// TwinCAT 3 PLC project PLC01
// ProgramVersion: 3.1.4026.16
// CompilerDefines: VISU_USEPROPERTYINFO
// libraries:
//   Tc2_Standard, * (Beckhoff Automation GmbH)
//   Tc2_System, * (Beckhoff Automation GmbH)
//   Tc2_Utilities, * (Beckhoff Automation GmbH)
//   Tc3_EventLogger, * (Beckhoff Automation GmbH)
//   VisuElemEventTable, * (System)
// project tree:
//   / GlobalTextList.TcGTLO, PlcTask.TcTTO, Visualization Manager.TcVMO (not stored)
//   POUs/ MAIN.TcPOU, prgAlarmHnd.TcPOU
//   VISUs/ Footer.TcVIS, Visualization.TcVIS
// real-time tasks:
//   TASK PlcTask: cycle T#10ms, priority 20, ADS port 350

CONFIGURATION PLC01
    RESOURCE PLC ON TwinCAT3
        TASK PlcTask(INTERVAL := T#10ms, PRIORITY := 20);
        PROGRAM MAIN WITH PlcTask : MAIN;
    END_RESOURCE
END_CONFIGURATION

// ---- POUs/MAIN.TcPOU
PROGRAM MAIN
VAR
END_VAR


prgAlarmHnd();

END_PROGRAM

// ---- POUs/prgAlarmHnd.TcPOU
PROGRAM prgAlarmHnd
VAR
	evtReader: FB_ReadTc3Events;
	actualEvts: ARRAY[1..80] OF ST_ReadEventW;
	histEvts: ARRAY[1..80] OF ST_ReadEventW;
	doClearEvts, doConfirmEvts, doRaiseEvt1, doRaiseEvt2, doRaiseEvt3, doClearTable:BOOL;
	alarm1, alarm2, alarm3: FB_TcAlarm;
	hr, hrLastErr: HRESULT;
	raiseEvt1Trig, raiseEvt2Trig, raiseEvt3Trig:R_TRIG;
	clearEvt1Trig, clearEvt2Trig, clearEvt3Trig: F_TRIG;
	doInitNow:BOOL:=TRUE;
END_VAR

IF doInitNow THEN
	hr := alarm1.CreateEx(TC_Events.UserAlarms.evt01,TRUE,0);
	IF failed(hr) THEN
		hrLastErr:=hr;
	END_IF
	hr := alarm2.CreateEx(TC_Events.UserAlarms.evt02,TRUE,0);
	IF failed(hr) THEN
		hrLastErr:=hr;
	END_IF
	hr := alarm3.CreateEx(TC_Events.UserAlarms.evt03,TRUE,0);
	IF failed(hr) THEN
		hrLastErr:=hr;
	END_IF
	doInitNow:=FALSE;
END_IF
raiseEvt1Trig(CLK:= doRaiseEvt1);
raiseEvt2Trig(CLK:= doRaiseEvt2);
raiseEvt3Trig(CLK:= doRaiseEvt3 );
clearEvt1Trig(CLK:= doRaiseEvt1);
clearEvt2Trig(CLK:= doRaiseEvt2);
clearEvt3Trig(CLK:= doRaiseEvt3);

IF raiseEvt1Trig.Q THEN
	alarm1.Raise(0);
END_IF
IF raiseEvt2Trig.Q THEN
	alarm2.Raise(0);
END_IF
IF raiseEvt3trig.Q THEN
	alarm3.Raise(0);
END_IF
IF clearEvt1Trig.Q THEN
	alarm1.Clear(0,FALSE);
END_IF
IF clearEvt2Trig.Q THEN
	alarm2.Clear(0,FALSE);
END_IF
IF clearEvt3Trig.Q THEN
	alarm3.Clear(0,FALSE);
END_IF
IF doConfirmEvts THEN
	alarm1.Confirm(0);
	alarm2.Confirm(0);
	alarm3.Confirm(0);
END_IF

evtReader(
	bReadEvents:= TRUE, 
	nLanguageID:=1031 , 
	eDateAndTimeFormat:=E_DateAndTimeFormat.de_DE , 
	bClearTable:= doClearTable, 
	eMinSeverity:= , 
	aEvents=>actualEvts , 
	nNumberOfEvents=> , 
	bError=> , 
	hrErrorCode=> );

END_PROGRAM

// ---- GlobalTextList.TcGTLO
TEXTLIST GlobalTextList
  989 = 'Alarme 1'
  381 = 'Alarme 2'
  386 = 'Alarmes'
  56 = 'Classe'
  849 = 'Clear'
  728 = 'Confirma'
  493 = 'Confirmado'
  120 = 'Dara'
  682 = 'Data'
  44 = 'Fonte'
  901 = 'Histórico'
  39 = 'Hora'
  829 = 'Id'
  14 = 'Limpa'
  587 = 'Mensagem'
  374 = 'Origem'
  83 = 'srcId'
END_TEXTLIST

// ---- VISUs/Footer.TcVIS
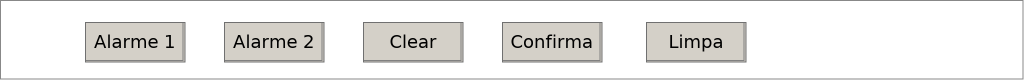
VISUALIZATION Footer  // 1024x80
    Button (85,22 100x40), "Alarme 1"
        toggle prgAlarmHnd.doRaiseEvt1
    Button (224,22 100x40), "Alarme 2"
        toggle prgAlarmHnd.doRaiseEvt2
    Button (363,22 100x40), "Clear"
        tap prgAlarmHnd.doClearEvts
    Button (502,22 100x40), "Confirma"
        tap prgAlarmHnd.doConfirmEvts
    Button (646,22 100x40), "Limpa"
        tap prgAlarmHnd.doClearTable
END_VISUALIZATION

// ---- VISUs/Visualization.TcVIS
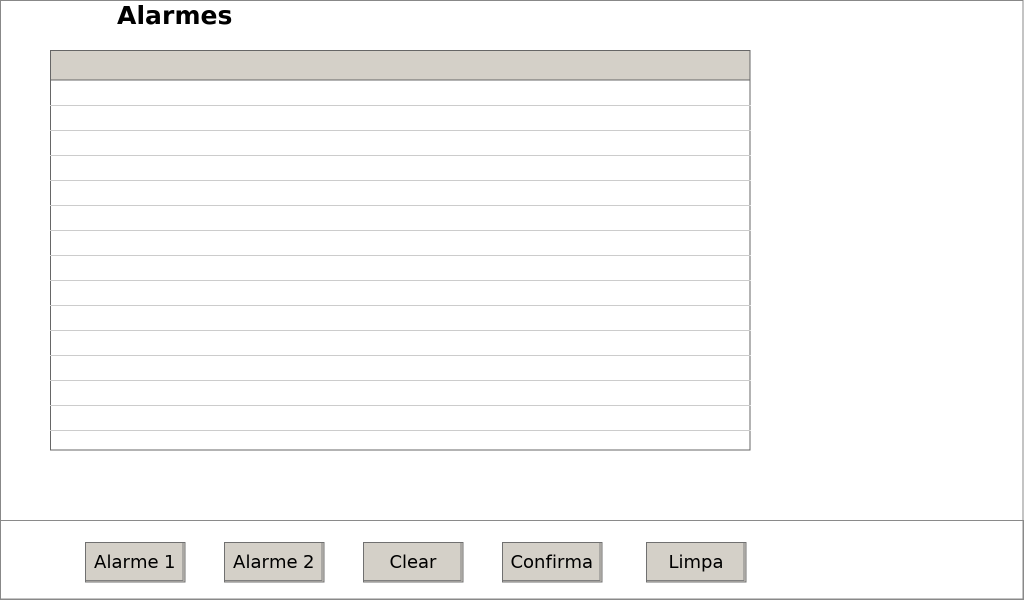
VISUALIZATION Visualization  // 1024x600
    Table (50,50 700x400), data array: prgAlarmHnd.actualEvts
        p3854506369: prgAlarmHnd.actualEvts[INDEX].nSourceID
        p1892666644: prgAlarmHnd.actualEvts[INDEX].nEventID
        p338671338: prgAlarmHnd.actualEvts[INDEX].nClass
        p2170511999: prgAlarmHnd.actualEvts[INDEX].nConfirmState
        p3723444502: prgAlarmHnd.actualEvts[INDEX].nResetState
        p1218418051: prgAlarmHnd.actualEvts[INDEX].sSource
        p746581629: prgAlarmHnd.actualEvts[INDEX].sDate
        p3104783080: prgAlarmHnd.actualEvts[INDEX].sTime
        p2501879983: prgAlarmHnd.actualEvts[INDEX].sComputer
        p7306298: prgAlarmHnd.actualEvts[INDEX].sMessageText
        p1933151965: prgAlarmHnd.actualEvts[INDEX].bQuitMessage
        p3863566920: prgAlarmHnd.actualEvts[INDEX].bConfirmable
        p1755163831: Classe
        p505689113: Origem
        p1757482276: Data
        p4088588272: Hora
        p516019884: Mensagem
        p1014161805: 80 - 1 + INT#1
    Label (100,0 150x30), "Alarmes"
    Frame (0,520 1024x80)
        shows Footer()
END_VISUALIZATION
